FUNCTION_BLOCK FB_WatchPhotoelectricBarrier
VAR_INPUT
	nInterrupted		: UINT;
END_VAR
VAR_OUTPUT
	bInterrupted		: BOOL;
END_VAR

IF nInterrupted < (32767 / 2) THEN
	bInterrupted := TRUE;
ELSE
	bInterrupted := FALSE;
END_IF

END_FUNCTION_BLOCK

(* stored: Version 1.1.0.1, ProductVersion 3.1.4024.11
   POU FB_WatchPhotoelectricBarrier: Id {7e558642-c1c0-44b6-9acf-d677532fb110}, SpecialFunc None *)
